Staubli VAL3: remTest.pgx

program remTest(string& sArgs[] (dimensions=1), string& sReturn[] (dimensions=1))
  local bool bOk
  local num nAzi
  local num nEle
  local num nLoop
  local num nRX
  local num nRY
  local num nRad
  local num nVal
  local num nX
  local num nY
  local num nZ
  local string sArgsLoop
  local trsf trCalc
  local trsf trTrans
begin
  //Misc current test
  nLoop=0
  sArgsLoop=sArgs
  while nLoop<3
    sArgsLoop=toNum(sArgsLoop,nVal,bOk)
    if bOk
      switch nLoop
        case 0
          nAzi=nVal
        break
        case 1
          nEle=nVal
        break
        case 2
          nRad=nVal
        break
      endSwitch
      nLoop=nLoop+1
    else
      call remErrNum("CMDTEST",sArgs,sReturn)
      return
    endIf
  endWhile

  nZ=nRad*cos(nEle)*cos(nAzi)
  nX=nRad*cos(nEle)*sin(nAzi)
  nY=nRad*sin(nEle)
  // Decide direction det is currently facing, keep det pointed to origin
  call remCalcHereSph()
  if abs(nRXHere+nElHere)<90
    nRX=-nEle
  else
    nRX=180-nEle
  endIf
  if abs(nRYHere+nAzHere)<90
    nRY=-nAzi
  else
    nRY=180-nAzi
  endIf
  trCalc={nX,nY,nZ,nRX,nRY,nRZHere}

  trTrans={0,0,0,0,0,0}
  trTrans=trTrans*{0,0,0,0,nAzi,0}
  trTrans=trTrans*{0,0,0,-nEle,0,0}
  trTrans=trTrans*{0,0,nRad,0,0,0}
  trTrans=trTrans*{0,0,0,-180,0,0}

  putln("trCalc:  "+toString(sNumConv,trCalc.x)+" "+toString(sNumConv,trCalc.y)+" "+toString(sNumConv,trCalc.z))
  putln("         "+toString(sNumConv,trCalc.rx)+" "+toString(sNumConv,trCalc.ry)+" "+toString(sNumConv,trCalc.rz))
  putln("trTrans: "+toString(sNumConv,trTrans.x)+" "+toString(sNumConv,trTrans.y)+" "+toString(sNumConv,trTrans.z))
  putln("         "+toString(sNumConv,trTrans.rx)+" "+toString(sNumConv,trTrans.ry)+" "+toString(sNumConv,trTrans.rz))

  sReturn="No output"
end
